// TIA Portal V17 export
// export: Created 2023-02-13T11:16:45.0045063Z, ExportSetting WithDefaults, DisplayName Totally Integrated Automation Portal, DisplayVersion V17, DisplayName TIA Portal Openness, DisplayVersion V17, DisplayName TIA Portal Teamcenter Gateway, DisplayVersion V17, DisplayName TIA Portal Version Control Interface, DisplayVersion V17, DisplayName SINAMICS Startdrive Advanced, DisplayVersion V17, DisplayName SINAMICS Startdrive G130, G150, S120, S150, SINAMICS MV, S210, DisplayVersion V17, DisplayName SINAMICS Startdrive G110M, G120, G120C, G120D, G120P, G115D, DisplayVersion V17, DisplayName STEP 7 Professional, DisplayVersion V17, DisplayName STEP 7 Safety, DisplayVersion V17, DisplayName WinCC Professional, DisplayVersion V17
ORGANIZATION_BLOCK "Main"   // OB1, LAD, ProgramCycle
TITLE = "Main Program Sweep (Cycle)"
{ S7_Optimized_Access := 'TRUE' }
VERSION : 0.1
// stored: AutoNumber true, IsIECCheckEnabled false, SetENOAutomatically false
   VAR_INPUT
      Initial_Call : Bool;   // Initial call of this OB
      Remanence : Bool;   // =True, if remanent data are available
   END_VAR
   VAR_TEMP   // added for the SCL form of the ladder/FBD networks
      _w1 : Bool;
      _w2 : Bool;
   END_VAR
BEGIN

REGION Network 1: Read Local date and time
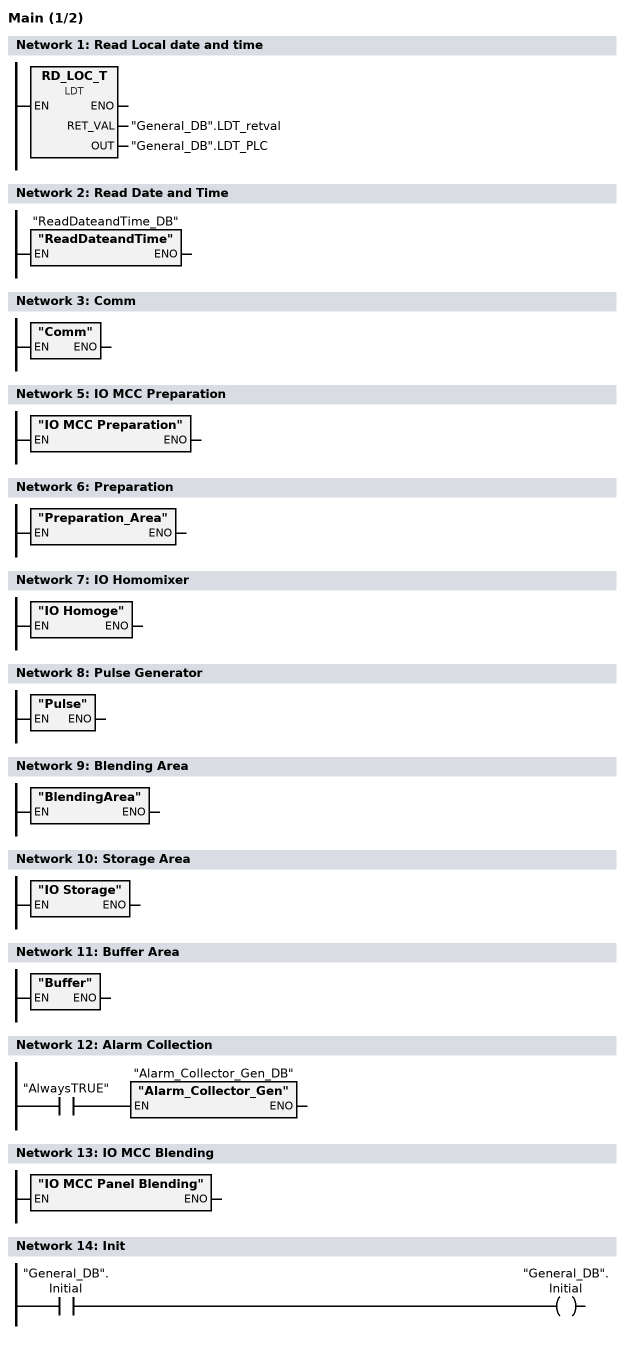
   RUNG wire#powerrail
      { S7_Templates := "date_type := LDT" } RD_LOC_T(RET_VAL => "General_DB".LDT_retval, OUT => "General_DB".LDT_PLC)
   END_RUNG
   // the same network as SCL:
   "General_DB".LDT_retval := RD_LOC_T(OUT => "General_DB".LDT_PLC);
END_REGION

REGION Network 2: Read Date and Time
   RUNG wire#powerrail
      "ReadDateandTime_DB"()
   END_RUNG
   // the same network as SCL:
   "ReadDateandTime_DB"();   // "ReadDateandTime"
END_REGION

REGION Network 3: Comm
   RUNG wire#powerrail
      "Comm"()
   END_RUNG
   // the same network as SCL:
   "Comm"();
END_REGION

REGION Network 5: IO MCC Preparation
   RUNG wire#powerrail
      "IO MCC Preparation"()
   END_RUNG
   // the same network as SCL:
   "IO MCC Preparation"();
END_REGION

REGION Network 6: Preparation
   RUNG wire#powerrail
      "Preparation_Area"()
   END_RUNG
   // the same network as SCL:
   "Preparation_Area"();
END_REGION

REGION Network 7: IO Homomixer
   RUNG wire#powerrail
      "IO Homoge"()
   END_RUNG
   // the same network as SCL:
   "IO Homoge"();
END_REGION

REGION Network 8: Pulse Generator
   RUNG wire#powerrail
      "Pulse"()
   END_RUNG
   // the same network as SCL:
   "Pulse"();
END_REGION

REGION Network 9: Blending Area
   RUNG wire#powerrail
      "BlendingArea"()
   END_RUNG
   // the same network as SCL:
   "BlendingArea"();
END_REGION

REGION Network 10: Storage Area
   RUNG wire#powerrail
      "IO Storage"()
   END_RUNG
   // the same network as SCL:
   "IO Storage"();
END_REGION

REGION Network 11: Buffer Area
   RUNG wire#powerrail
      "Buffer"()
   END_RUNG
   // the same network as SCL:
   "Buffer"();
END_REGION

REGION Network 12: Alarm Collection
   RUNG wire#powerrail
      Contact( "AlwaysTRUE" )
      "Alarm_Collector_Gen_DB"()
   END_RUNG
   // the same network as SCL:
   IF "AlwaysTRUE" THEN
       "Alarm_Collector_Gen_DB"();   // "Alarm_Collector_Gen"
   END_IF;
END_REGION

REGION Network 13: IO MCC Blending
   RUNG wire#powerrail
      "IO MCC Panel Blending"()
   END_RUNG
   // the same network as SCL:
   "IO MCC Panel Blending"();
END_REGION

REGION Network 14: Init
   RUNG wire#powerrail
      Contact( "General_DB".Initial )
      Coil( "General_DB".Initial )
   END_RUNG
   // the same network as SCL:
   "General_DB".Initial := "General_DB".Initial;
END_REGION

REGION Network 15: End Block Reset initial
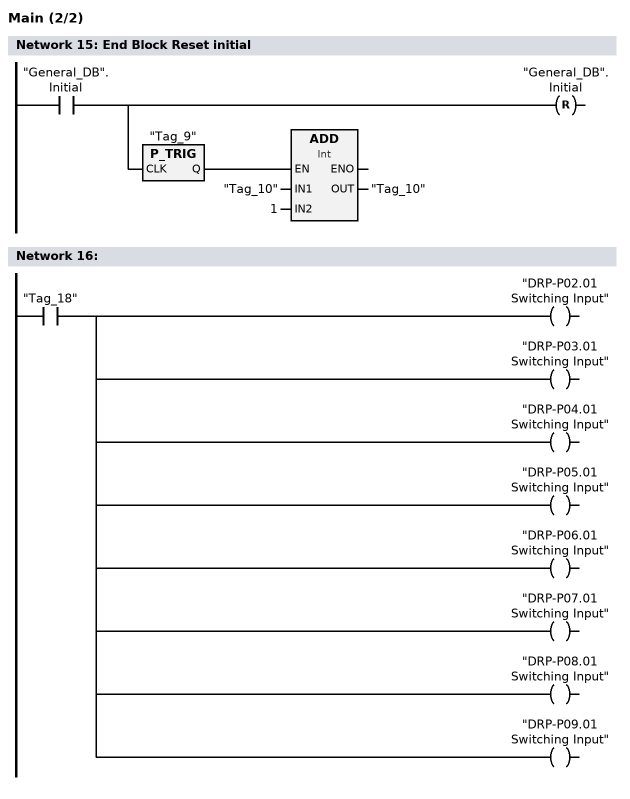
   RUNG wire#powerrail
      Contact( "General_DB".Initial )
      wire#w1
      R_Coil( "General_DB".Initial )
   END_RUNG
   RUNG wire#w1
      P_Trig( "Tag_9" )
      { S7_Templates := "SrcType := Int" } Add(in1 := "Tag_10", in2 := 1, out => "Tag_10")
   END_RUNG
   // the same network as SCL:
   #_w1 := "General_DB".Initial;
   IF #_w1 THEN "General_DB".Initial := FALSE; END_IF;
   #_w2 := #_w1 AND NOT "Tag_9";   // rising edge
   "Tag_9" := #_w1;
   IF #_w2 THEN "Tag_10" := "Tag_10" + 1; END_IF;
END_REGION

REGION Network 16
   RUNG wire#powerrail
      Contact( "Tag_18" )
      wire#w1
      Coil( "DRP-P02.01 Switching Input" )
   END_RUNG
   RUNG wire#w1
      Coil( "DRP-P03.01 Switching Input" )
   END_RUNG
   RUNG wire#w1
      Coil( "DRP-P04.01 Switching Input" )
   END_RUNG
   RUNG wire#w1
      Coil( "DRP-P05.01 Switching Input" )
   END_RUNG
   RUNG wire#w1
      Coil( "DRP-P06.01 Switching Input" )
   END_RUNG
   RUNG wire#w1
      Coil( "DRP-P07.01 Switching Input" )
   END_RUNG
   RUNG wire#w1
      Coil( "DRP-P08.01 Switching Input" )
   END_RUNG
   RUNG wire#w1
      Coil( "DRP-P09.01 Switching Input" )
   END_RUNG
   // the same network as SCL:
   "DRP-P02.01 Switching Input" := "Tag_18";
   "DRP-P03.01 Switching Input" := "Tag_18";
   "DRP-P04.01 Switching Input" := "Tag_18";
   "DRP-P05.01 Switching Input" := "Tag_18";
   "DRP-P06.01 Switching Input" := "Tag_18";
   "DRP-P07.01 Switching Input" := "Tag_18";
   "DRP-P08.01 Switching Input" := "Tag_18";
   "DRP-P09.01 Switching Input" := "Tag_18";
END_REGION
END_ORGANIZATION_BLOCK
